GLOBALCONSTANTS AID_GD (* Graphic data (PNG) object attribute ids *)
  (* Standard: 61499-1; Description: Copyright (c) 2023 HR Agrartechnik GmbH This program and the accompanying materials are made available under the terms of the Eclipse Public License 2.0 which is available at https://www.eclipse.org/legal/epl-2.0/ SPDX-License-Identifier: EPL-2.0 *)
  (* Version 1.0, 2026-06-20, Franz Höpfinger, HR Agrartechnik GmbH *)
  PACKAGE isobus::UT::Q::const::AID;
  IMPORT eclipse4diac::core::TypeHash;
  VAR_GLOBAL CONSTANT
    FORMAT : USINT := USINT#1; (* 1: AID_GD_FORMAT - Graphic type: 0 = PNG, restricted to 32bit RGBA maximum. *)
  END_VAR
END_GLOBALCONSTANTS
